Fanuc KAREL source: kc00040.KL

-- PROVISIONAL review KL for V940-1; original PC SHA256 ba2ce702cb52c58b8121dfb237800881a84b93cf478b3186c7234ecc1938b25d
-- Incomplete behavior may be omitted. Consult companion uncertainty JSON. Do not deploy.
PROGRAM KC00040
%NOLOCKGROUP
BEGIN
  -- V9_ZERO_TABLE_METADATA_HINT layout=0002_ascii; no indexed target words; source/name/runtime held
  -- UNRESOLVED_PC offsets 5-33; opcodes 27,22,22,22,22,31
  -- UNRESOLVED_PC offsets 38-42; opcodes 7F
END KC00040
